PROGRAM P3_01_SP_BatchData
VAR
END_VAR
VAR // added by the converter: edge detectors and wires of the graphical bodies
    _rt1, _rt2 : R_TRIG;
END_VAR

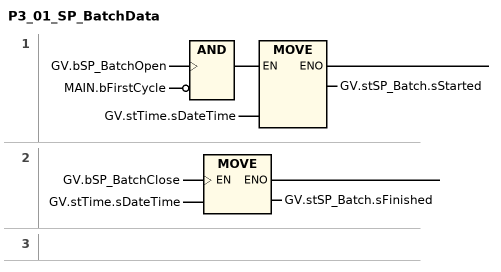
// NETWORK 1
_rt1(CLK := GV.bSP_BatchOpen);
IF _rt1.Q AND NOT MAIN.bFirstCycle THEN GV.stSP_Batch.sStarted := GV.stTime.sDateTime; END_IF

// NETWORK 2
_rt2(CLK := GV.bSP_BatchClose);
IF _rt2.Q THEN GV.stSP_Batch.sFinished := GV.stTime.sDateTime; END_IF

// NETWORK 3

END_PROGRAM

(* stored: Version 1.1.0.1, ProductVersion 3.1.4024.12
   POU P3_01_SP_BatchData: Id {0f1dfd81-2b63-4010-81db-c491f388e45c}, SpecialFunc None *)
